SYSTEM TestSystem (* System Configuration *)
  (* Standard: 61499-1 *)
  (* Version 0.3, 2003-12-05, JHC, Rockwell Automation, Renamed from NEWSYSTEM. *)
  (* Version 0.2, 2002-11-05, JHC, Rockwell Automation, Fixed missing (empty) FBD in Application. *)
  (* Version 0.1, 2002-01-17, JHC, Rockwell Automation, Minor cleanup *)
  (* Version 0.0, 2000-05-27, JHC, Rockwell Automation *)
  APPLICATION APP1
  END_APPLICATION
  DEVICE View : FRAME_DEVICE(BOUNDS := [100,100,200,100])
    RESOURCE viewPanel : PANEL_RESOURCE
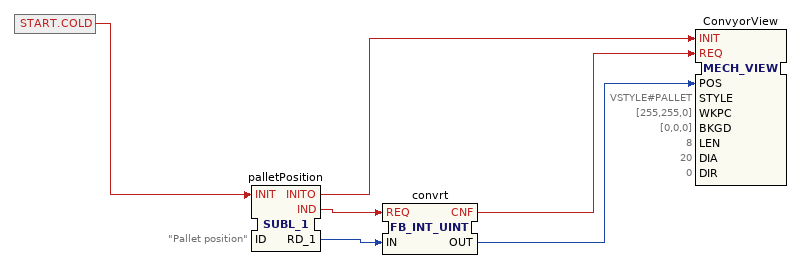
      FBS
        ConvyorView : MECH_VIEW(STYLE := VSTYLE#PALLET, WKPC := [255,255,0], BKGD := [0,0,0], LEN := 8, DIA := 20, DIR := 0);
        palletPosition : SUBL_1(ID := "Pallet position");
        convrt : FB_INT_UINT;
      END_FBS
      EVENT_CONNECTIONS
        START.COLD TO palletPosition.INIT;
        palletPosition.INITO TO ConvyorView.INIT;
        palletPosition.IND TO convrt.REQ;
        convrt.CNF TO ConvyorView.REQ;
      END_CONNECTIONS
      DATA_CONNECTIONS
        palletPosition.RD_1 TO convrt.IN;
        convrt.OUT TO ConvyorView.POS;
      END_CONNECTIONS
    END_RESOURCE
  END_DEVICE
  DEVICE HMI : FRAME_DEVICE(BOUNDS := [300,100,200,100])
    RESOURCE hmiPanel : PANEL_RESOURCE
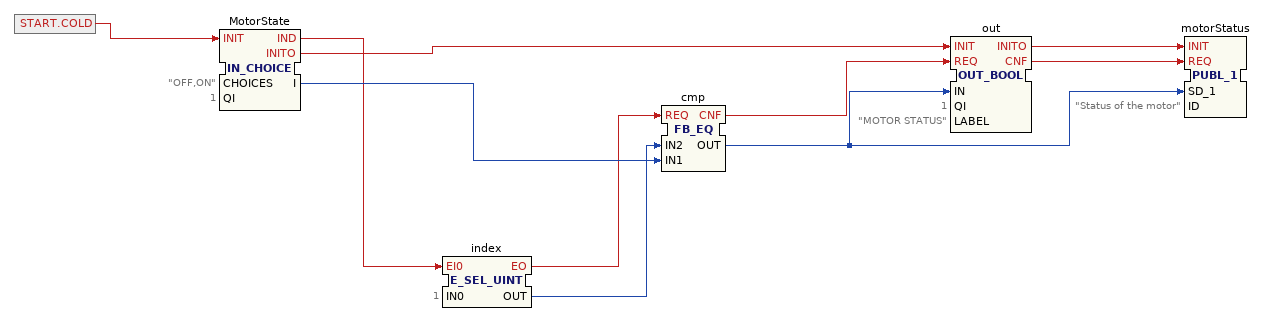
      FBS
        out : OUT_BOOL(QI := 1, LABEL := "MOTOR STATUS");
        MotorState : IN_CHOICE(CHOICES := "OFF,ON", QI := 1);
        index : E_SEL_UINT(IN0 := 1);
        cmp : FB_EQ;
        motorStatus : PUBL_1(ID := "Status of the motor");
      END_FBS
      EVENT_CONNECTIONS
        START.COLD TO MotorState.INIT;
        MotorState.IND TO index.EI0;
        MotorState.INITO TO out.INIT;
        index.EO TO cmp.REQ;
        cmp.CNF TO out.REQ;
        out.INITO TO motorStatus.INIT;
        out.CNF TO motorStatus.REQ;
      END_CONNECTIONS
      DATA_CONNECTIONS
        index.OUT TO cmp.IN2;
        MotorState.I TO cmp.IN1;
        cmp.OUT TO out.IN;
        cmp.OUT TO motorStatus.SD_1;
      END_CONNECTIONS
    END_RESOURCE
  END_DEVICE
  DEVICE Model : FRAME_DEVICE(BOUNDS := [200,200,100,100] (* Model that checks the status of the motor. *))
    RESOURCE modelPanel : PANEL_RESOURCE
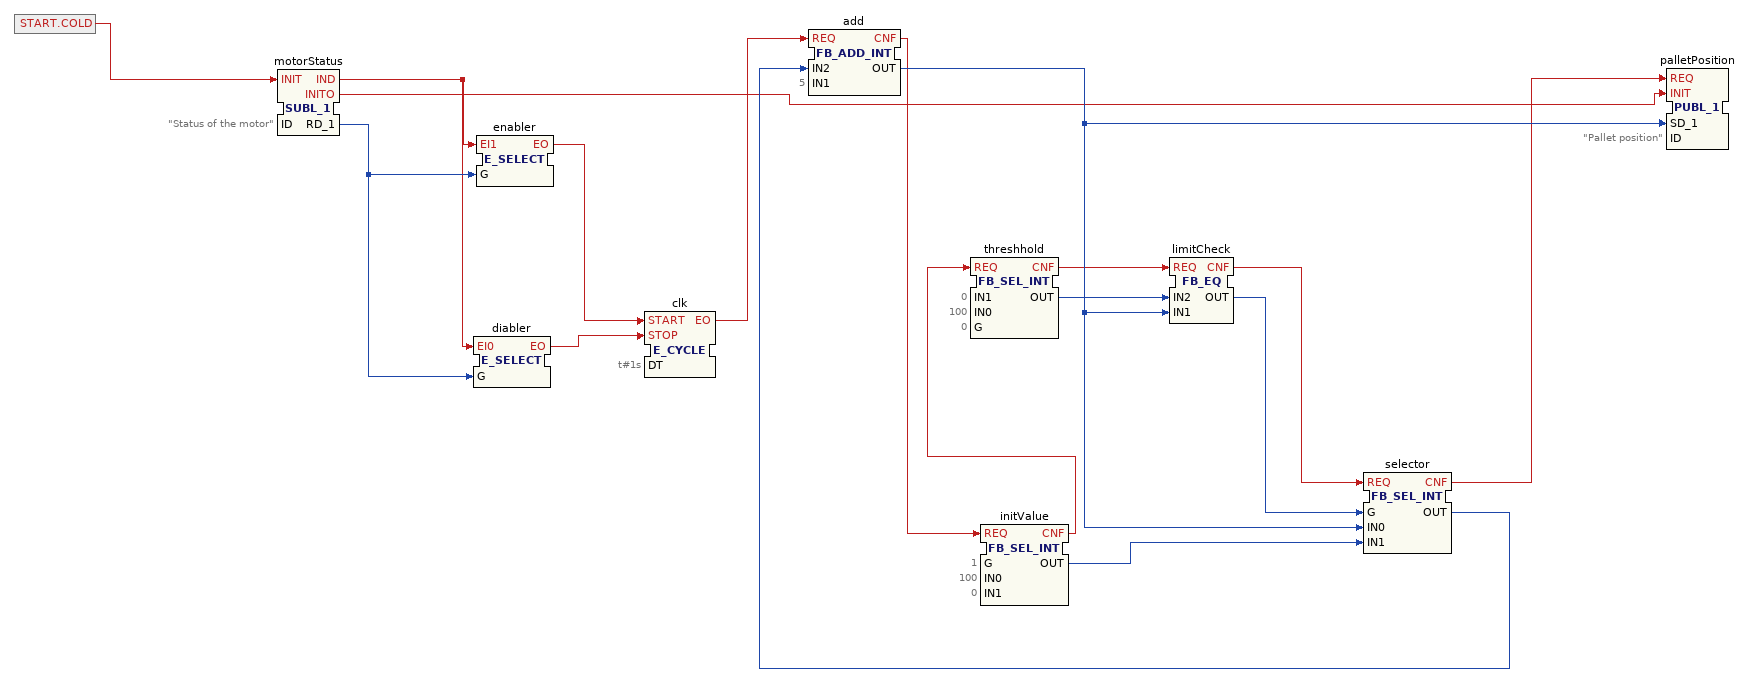
      FBS
        motorStatus : SUBL_1(ID := "Status of the motor");
        add : FB_ADD_INT(IN1 := 5);
        enabler : E_SELECT;
        palletPosition : PUBL_1(ID := "Pallet position");
        clk : E_CYCLE(DT := t#1s);
        diabler : E_SELECT;
        limitCheck : FB_EQ;
        threshhold : FB_SEL_INT(IN1 := 0, IN0 := 100, G := 0);
        selector : FB_SEL_INT;
        initValue : FB_SEL_INT(G := 1, IN0 := 100, IN1 := 0);
      END_FBS
      EVENT_CONNECTIONS
        START.COLD TO motorStatus.INIT;
        enabler.EO TO clk.START;
        clk.EO TO add.REQ;
        diabler.EO TO clk.STOP;
        motorStatus.IND TO enabler.EI1;
        motorStatus.IND TO diabler.EI0;
        threshhold.CNF TO limitCheck.REQ;
        limitCheck.CNF TO selector.REQ;
        selector.CNF TO palletPosition.REQ;
        motorStatus.INITO TO palletPosition.INIT;
        add.CNF TO initValue.REQ;
        initValue.CNF TO threshhold.REQ;
      END_CONNECTIONS
      DATA_CONNECTIONS
        motorStatus.RD_1 TO enabler.G;
        add.OUT TO palletPosition.SD_1;
        motorStatus.RD_1 TO diabler.G;
        threshhold.OUT TO limitCheck.IN2;
        add.OUT TO limitCheck.IN1;
        limitCheck.OUT TO selector.G;
        add.OUT TO selector.IN0;
        selector.OUT TO add.IN2;
        initValue.OUT TO selector.IN1;
      END_CONNECTIONS
    END_RESOURCE
  END_DEVICE
END_SYSTEM
